FUNCTION_BLOCK SM_LinearVelocity
VAR_INPUT
	///New velocity value in millimeters per second
	{attribute 'OPC.UA.DA' := '0'}
	newMillimetersPerSecondValue: LREAL;
END_VAR
VAR_OUTPUT
	///Current status description
	{attribute 'OPC.UA.DA' := '1'}
	{attribute 'OPC.UA.DA.Access' := '1'}
	actualStatus: STRING;
	///Angular velocity in radians per second
	{attribute 'OPC.UA.DA' := '1'}
	{attribute 'OPC.UA.DA.Access' := '1'}
	millimetersPerSecond: QuantityValue;
END_VAR
VAR_IN_OUT
END_VAR
VAR
END_VAR

millimetersPerSecond(
    value := newMillimetersPerSecondValue,
    unit := Units.MILLIMETERS_PER_SECOND);

END_FUNCTION_BLOCK

(* stored: Version 1.1.0.1, ProductVersion 3.1.4019.2
   POU SM_LinearVelocity: Id {4e2eafa7-c416-428c-910b-7a62529221d8}, SpecialFunc None *)
